// TIA Portal V19 export
FUNCTION "Servo_PLS_Styring" : Void   // FC5, LAD
{ S7_Optimized_Access := 'TRUE' }
// stored: SetENOAutomatically false
BEGIN

REGION Network 1
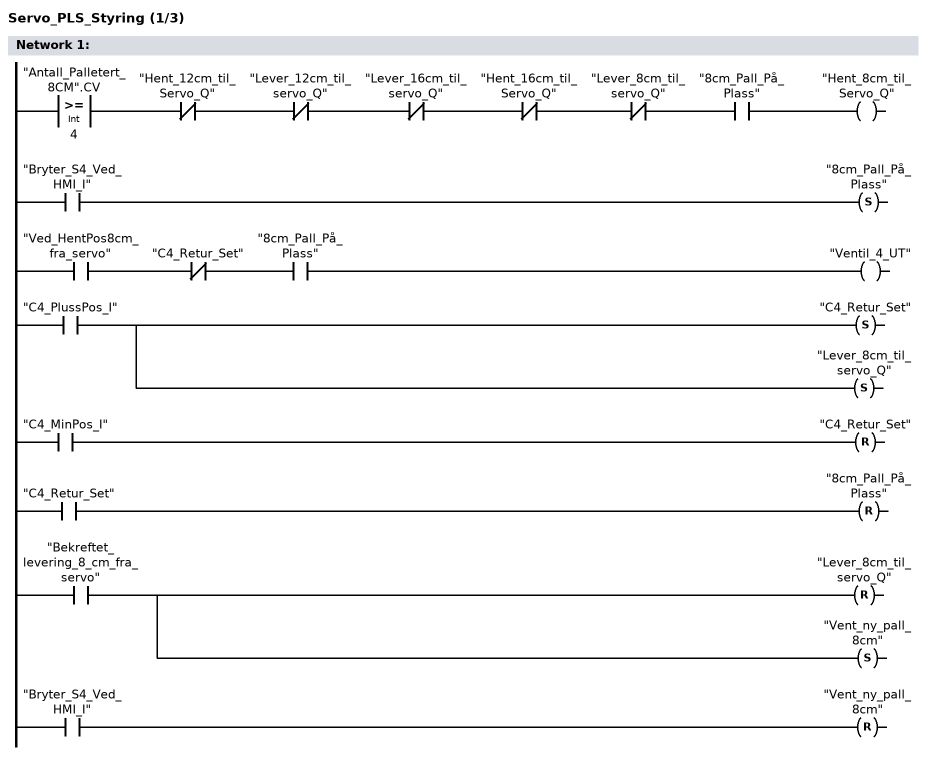
   RUNG wire#powerrail
      { S7_Templates := "SrcType := Int" } GE_Contact(in1 := "Antall_Palletert_8CM".CV, in2 := 4)
      I_Contact( "Hent_12cm_til_Servo_Q" )
      I_Contact( "Lever_12cm_til_servo_Q" )
      I_Contact( "Lever_16cm_til_servo_Q" )
      I_Contact( "Hent_16cm_til_Servo_Q" )
      I_Contact( "Lever_8cm_til_servo_Q" )
      Contact( "8cm_Pall_På_Plass" )
      Coil( "Hent_8cm_til_Servo_Q" )
   END_RUNG
   RUNG wire#powerrail
      Contact( "Bryter_S4_Ved_HMI_I" )
      S_Coil( "8cm_Pall_På_Plass" )
   END_RUNG
   RUNG wire#powerrail
      Contact( "Ved_HentPos8cm_fra_servo" )
      I_Contact( "C4_Retur_Set" )
      Contact( "8cm_Pall_På_Plass" )
      Coil( "Ventil_4_UT" )
   END_RUNG
   RUNG wire#powerrail
      Contact( "C4_PlussPos_I" )
      wire#w1
      S_Coil( "C4_Retur_Set" )
   END_RUNG
   RUNG wire#w1
      S_Coil( "Lever_8cm_til_servo_Q" )
   END_RUNG
   RUNG wire#powerrail
      Contact( "C4_MinPos_I" )
      R_Coil( "C4_Retur_Set" )
   END_RUNG
   RUNG wire#powerrail
      Contact( "C4_Retur_Set" )
      R_Coil( "8cm_Pall_På_Plass" )
   END_RUNG
   RUNG wire#powerrail
      Contact( "Bekreftet_levering_8_cm_fra_servo" )
      wire#w2
      R_Coil( "Lever_8cm_til_servo_Q" )
   END_RUNG
   RUNG wire#w2
      S_Coil( "Vent_ny_pall_8cm" )
   END_RUNG
   RUNG wire#powerrail
      Contact( "Bryter_S4_Ved_HMI_I" )
      R_Coil( "Vent_ny_pall_8cm" )
   END_RUNG
   // the same network as SCL:
   "Hent_8cm_til_Servo_Q" := ("Antall_Palletert_8CM".CV >= 4) AND NOT "Hent_12cm_til_Servo_Q" AND NOT "Lever_12cm_til_servo_Q" AND NOT "Lever_16cm_til_servo_Q" AND NOT "Hent_16cm_til_Servo_Q" AND NOT "Lever_8cm_til_servo_Q" AND "8cm_Pall_På_Plass";
   IF "Bryter_S4_Ved_HMI_I" THEN "8cm_Pall_På_Plass" := TRUE; END_IF;
   "Ventil_4_UT" := "Ved_HentPos8cm_fra_servo" AND NOT "C4_Retur_Set" AND "8cm_Pall_På_Plass";
   IF "C4_PlussPos_I" THEN
       "C4_Retur_Set" := TRUE;
       "Lever_8cm_til_servo_Q" := TRUE;
   END_IF;
   IF "C4_MinPos_I" THEN "C4_Retur_Set" := FALSE; END_IF;
   IF "C4_Retur_Set" THEN "8cm_Pall_På_Plass" := FALSE; END_IF;
   IF "Bekreftet_levering_8_cm_fra_servo" THEN
       "Lever_8cm_til_servo_Q" := FALSE;
       "Vent_ny_pall_8cm" := TRUE;
   END_IF;
   IF "Bryter_S4_Ved_HMI_I" THEN "Vent_ny_pall_8cm" := FALSE; END_IF;
END_REGION

REGION Network 2
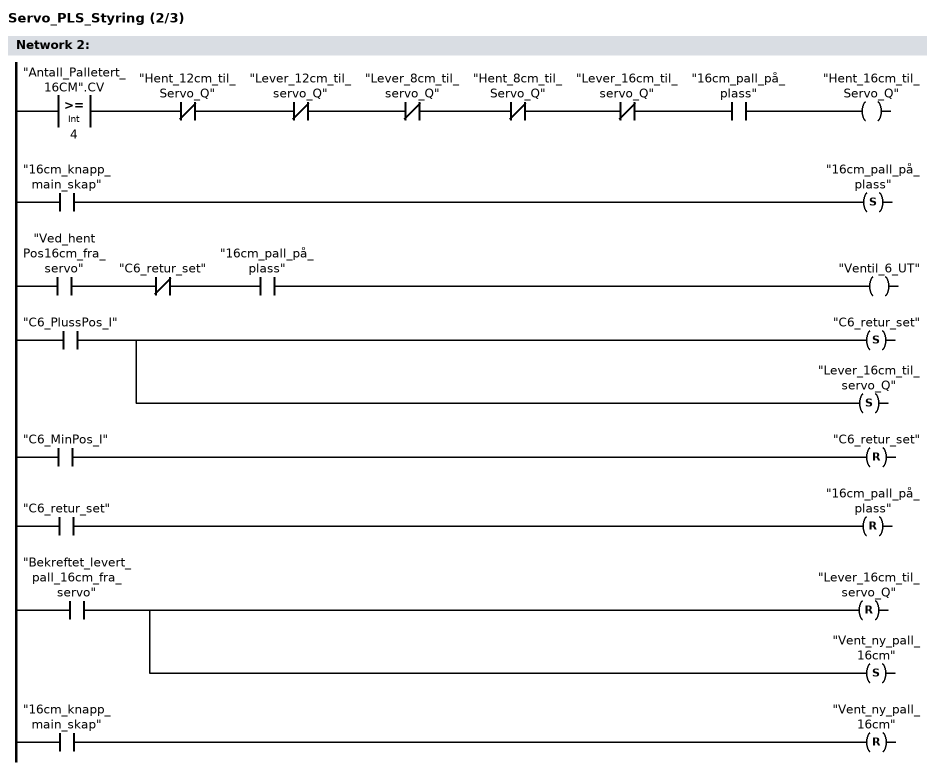
   RUNG wire#powerrail
      { S7_Templates := "SrcType := Int" } GE_Contact(in1 := "Antall_Palletert_16CM".CV, in2 := 4)
      I_Contact( "Hent_12cm_til_Servo_Q" )
      I_Contact( "Lever_12cm_til_servo_Q" )
      I_Contact( "Lever_8cm_til_servo_Q" )
      I_Contact( "Hent_8cm_til_Servo_Q" )
      I_Contact( "Lever_16cm_til_servo_Q" )
      Contact( "16cm_pall_på_plass" )
      Coil( "Hent_16cm_til_Servo_Q" )
   END_RUNG
   RUNG wire#powerrail
      Contact( "16cm_knapp_main_skap" )
      S_Coil( "16cm_pall_på_plass" )
   END_RUNG
   RUNG wire#powerrail
      Contact( "Ved_hentPos16cm_fra_servo" )
      I_Contact( "C6_retur_set" )
      Contact( "16cm_pall_på_plass" )
      Coil( "Ventil_6_UT" )
   END_RUNG
   RUNG wire#powerrail
      Contact( "C6_PlussPos_I" )
      wire#w1
      S_Coil( "C6_retur_set" )
   END_RUNG
   RUNG wire#w1
      S_Coil( "Lever_16cm_til_servo_Q" )
   END_RUNG
   RUNG wire#powerrail
      Contact( "C6_MinPos_I" )
      R_Coil( "C6_retur_set" )
   END_RUNG
   RUNG wire#powerrail
      Contact( "C6_retur_set" )
      R_Coil( "16cm_pall_på_plass" )
   END_RUNG
   RUNG wire#powerrail
      Contact( "Bekreftet_levert_pall_16cm_fra_servo" )
      wire#w2
      R_Coil( "Lever_16cm_til_servo_Q" )
   END_RUNG
   RUNG wire#w2
      S_Coil( "Vent_ny_pall_16cm" )
   END_RUNG
   RUNG wire#powerrail
      Contact( "16cm_knapp_main_skap" )
      R_Coil( "Vent_ny_pall_16cm" )
   END_RUNG
   // the same network as SCL:
   "Hent_16cm_til_Servo_Q" := ("Antall_Palletert_16CM".CV >= 4) AND NOT "Hent_12cm_til_Servo_Q" AND NOT "Lever_12cm_til_servo_Q" AND NOT "Lever_8cm_til_servo_Q" AND NOT "Hent_8cm_til_Servo_Q" AND NOT "Lever_16cm_til_servo_Q" AND "16cm_pall_på_plass";
   IF "16cm_knapp_main_skap" THEN "16cm_pall_på_plass" := TRUE; END_IF;
   "Ventil_6_UT" := "Ved_hentPos16cm_fra_servo" AND NOT "C6_retur_set" AND "16cm_pall_på_plass";
   IF "C6_PlussPos_I" THEN
       "C6_retur_set" := TRUE;
       "Lever_16cm_til_servo_Q" := TRUE;
   END_IF;
   IF "C6_MinPos_I" THEN "C6_retur_set" := FALSE; END_IF;
   IF "C6_retur_set" THEN "16cm_pall_på_plass" := FALSE; END_IF;
   IF "Bekreftet_levert_pall_16cm_fra_servo" THEN
       "Lever_16cm_til_servo_Q" := FALSE;
       "Vent_ny_pall_16cm" := TRUE;
   END_IF;
   IF "16cm_knapp_main_skap" THEN "Vent_ny_pall_16cm" := FALSE; END_IF;
END_REGION

REGION Network 3
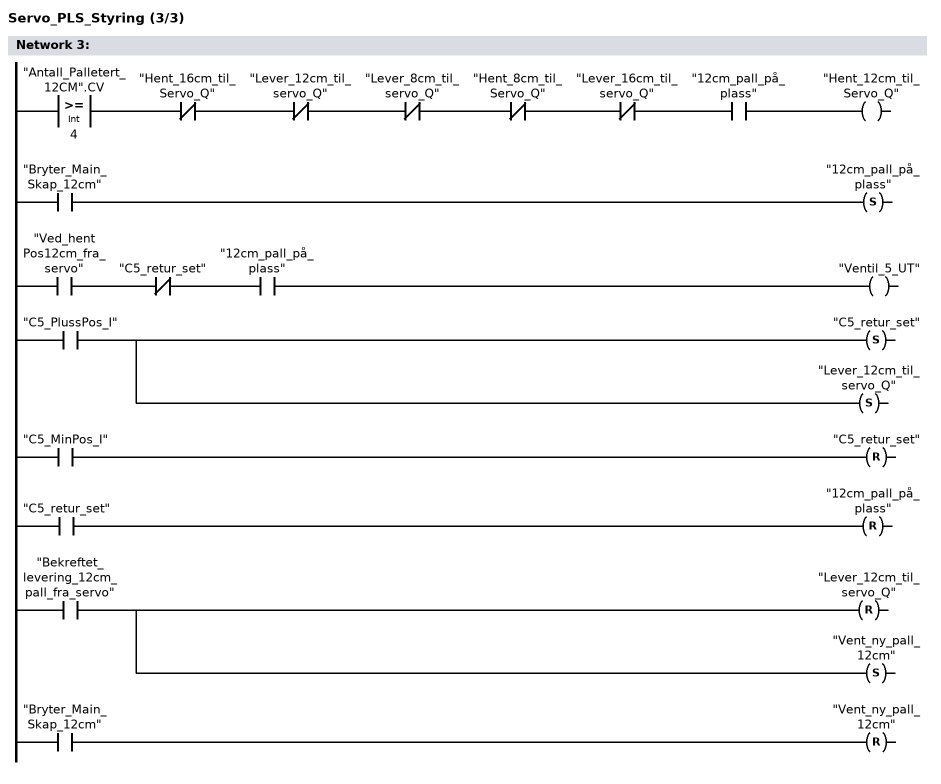
   RUNG wire#powerrail
      { S7_Templates := "SrcType := Int" } GE_Contact(in1 := "Antall_Palletert_12CM".CV, in2 := 4)
      I_Contact( "Hent_16cm_til_Servo_Q" )
      I_Contact( "Lever_12cm_til_servo_Q" )
      I_Contact( "Lever_8cm_til_servo_Q" )
      I_Contact( "Hent_8cm_til_Servo_Q" )
      I_Contact( "Lever_16cm_til_servo_Q" )
      Contact( "12cm_pall_på_plass" )
      Coil( "Hent_12cm_til_Servo_Q" )
   END_RUNG
   RUNG wire#powerrail
      Contact( "Bryter_Main_Skap_12cm" )
      S_Coil( "12cm_pall_på_plass" )
   END_RUNG
   RUNG wire#powerrail
      Contact( "Ved_hentPos12cm_fra_servo" )
      I_Contact( "C5_retur_set" )
      Contact( "12cm_pall_på_plass" )
      Coil( "Ventil_5_UT" )
   END_RUNG
   RUNG wire#powerrail
      Contact( "C5_PlussPos_I" )
      wire#w1
      S_Coil( "C5_retur_set" )
   END_RUNG
   RUNG wire#w1
      S_Coil( "Lever_12cm_til_servo_Q" )
   END_RUNG
   RUNG wire#powerrail
      Contact( "C5_MinPos_I" )
      R_Coil( "C5_retur_set" )
   END_RUNG
   RUNG wire#powerrail
      Contact( "C5_retur_set" )
      R_Coil( "12cm_pall_på_plass" )
   END_RUNG
   RUNG wire#powerrail
      Contact( "Bekreftet_levering_12cm_pall_fra_servo" )
      wire#w2
      R_Coil( "Lever_12cm_til_servo_Q" )
   END_RUNG
   RUNG wire#w2
      S_Coil( "Vent_ny_pall_12cm" )
   END_RUNG
   RUNG wire#powerrail
      Contact( "Bryter_Main_Skap_12cm" )
      R_Coil( "Vent_ny_pall_12cm" )
   END_RUNG
   // the same network as SCL:
   "Hent_12cm_til_Servo_Q" := ("Antall_Palletert_12CM".CV >= 4) AND NOT "Hent_16cm_til_Servo_Q" AND NOT "Lever_12cm_til_servo_Q" AND NOT "Lever_8cm_til_servo_Q" AND NOT "Hent_8cm_til_Servo_Q" AND NOT "Lever_16cm_til_servo_Q" AND "12cm_pall_på_plass";
   IF "Bryter_Main_Skap_12cm" THEN "12cm_pall_på_plass" := TRUE; END_IF;
   "Ventil_5_UT" := "Ved_hentPos12cm_fra_servo" AND NOT "C5_retur_set" AND "12cm_pall_på_plass";
   IF "C5_PlussPos_I" THEN
       "C5_retur_set" := TRUE;
       "Lever_12cm_til_servo_Q" := TRUE;
   END_IF;
   IF "C5_MinPos_I" THEN "C5_retur_set" := FALSE; END_IF;
   IF "C5_retur_set" THEN "12cm_pall_på_plass" := FALSE; END_IF;
   IF "Bekreftet_levering_12cm_pall_fra_servo" THEN
       "Lever_12cm_til_servo_Q" := FALSE;
       "Vent_ny_pall_12cm" := TRUE;
   END_IF;
   IF "Bryter_Main_Skap_12cm" THEN "Vent_ny_pall_12cm" := FALSE; END_IF;
END_REGION
END_FUNCTION
